{attribute 'qualified_only'}
{attribute 'strict'}
TYPE E_States :
(
	eStop := 0,
	eMovingLeft,
	eMovingRight
);
END_TYPE

(* stored: Version 1.1.0.1, ProductVersion 3.1.4024.12
   DUT E_States: Id {c0e4076b-9a29-479c-884c-bd0495ebedb7} *)
